FUNCTION_BLOCK T_SubModuleCollection EXTENDS T_CollectionBase

METHOD PUBLIC AddModule : BOOL
VAR_INPUT
  newModule : I_PackML_BaseModule;
END_VAR
VAR
	item : I_InterfaceBase;
END_VAR
IF newModule = 0 THEN
	LogError( 'Cannot AddModule invalid ref' );
	RETURN;
END_IF

IF NOT __QUERYINTERFACE(newModule, item) THEN
	LogError( 'Cannot AddModule  NOT __QUERYINTERFACE(newComponent, item)' );
	RETURN;
END_IF

IF HasItem( item := item ) THEN
	LogWarning( 'Module already in collection.' );
	RETURN;
END_IF

AddModule := addInSpareSlot( item := item );
END_METHOD

METHOD PUBLIC AllInAskedState : BOOL
VAR_INPUT
	State : Tc3_PackML_V2.E_PMLState;
END_VAR
VAR
	i : UDINT;
	Module : I_PackML_BaseModule;
	item : I_InterfaceBase;
END_VAR
IF Count = 0 THEN
	AllInAskedState := TRUE;
	RETURN;
END_IF

FOR i := 0 TO Count -1 DO

	IF NOT 	TryGetItem(i, item => item) THEN
		RETURN;
	END_IF
	
	IF NOT __QUERYINTERFACE(item, Module) THEN
		RETURN;
	END_IF
		
	IF Module.CurrentState <> State THEN
		RETURN;
	END_IF
		
END_FOR

AllInAskedState := TRUE;
END_METHOD

PROPERTY AnyError : BOOL
GET
VAR
  i : UDINT;
  Module : I_PackML_BaseModule;
  item : I_InterfaceBase;
 END_VAR
IF Count = 0 THEN
  RETURN;
END_IF

FOR i := 0 TO Count -1 DO

	IF NOT 	TryGetItem(i, item => item) THEN
		RETURN;
	END_IF
	
	IF NOT __QUERYINTERFACE(item, Module) THEN
		RETURN;
	END_IF
		
	IF Module.Error THEN
		AnyError := TRUE;
		RETURN;
	END_IF

END_FOR
END_GET
END_PROPERTY

METHOD PUBLIC AnyInAskedState : BOOL
VAR_INPUT
	State : Tc3_PackML_V2.E_PMLState;
END_VAR
VAR_OUTPUT
	Module : I_PackML_BaseModule;	
END_VAR
VAR
	i : UDINT;

	item : I_InterfaceBase;
END_VAR
IF Count = 0 THEN
	RETURN;
END_IF

FOR i := 0 TO Count -1 DO

	IF NOT 	TryGetItem(i, item => item) THEN
		RETURN;
	END_IF
	
	IF NOT __QUERYINTERFACE(item, Module) THEN
		RETURN;
	END_IF
		
	IF Module.CurrentState = State THEN
		AnyInAskedState := TRUE;
		RETURN;
	END_IF
		
END_FOR
END_METHOD

METHOD CyclicLogic
VAR
  i : UDINT;
  Module : I_PackML_BaseModule;
  item : I_InterfaceBase;
END_VAR
IF Count = 0 THEN
  RETURN;
END_IF

FOR i := 0 TO Count -1 DO
	TryGetItem(i, item => item);
	__QUERYINTERFACE(item, Module);
	IF Module <> 0 THEN
  		Module.CyclicLogic();
	END_IF	
END_FOR
END_METHOD

PROPERTY PUBLIC InitialisedAll : BOOL
GET
VAR
  i : UDINT;
  Module : I_PackML_BaseModule;
  item : I_InterfaceBase;
 END_VAR
IF Count = 0 THEN
	InitialisedAll := TRUE;
  RETURN;
END_IF

FOR i := 0 TO Count -1 DO

	IF NOT 	TryGetItem(i, item => item) THEN
		RETURN;
	END_IF
	
	IF NOT __QUERYINTERFACE(item, Module) THEN
		RETURN;
	END_IF
		
	IF NOT Module.InitComplete THEN
		RETURN;
	END_IF
		

END_FOR

InitialisedAll := TRUE;
END_GET
END_PROPERTY

METHOD PUBLIC NotifyModeChanged
VAR_INPUT
    Mode : E_PMLUnitMode;
END_VAR
VAR
	i : UDINT;
	Module : I_PackML_BaseModule;
	item : I_InterfaceBase;
END_VAR
IF Count = 0 THEN
  RETURN;
END_IF

FOR i := 0 TO Count -1 DO

	IF NOT 	TryGetItem(i, item => item) THEN
		RETURN;
	END_IF
	
	IF NOT __QUERYINTERFACE(item, Module) THEN
		RETURN;
	END_IF
		
	Module.ChangeMode(Mode);
		
END_FOR
END_METHOD

METHOD PUBLIC NotifyStateChanged
VAR_INPUT
	CommandedState : Tc3_PackML_V2.E_PMLCommand;
END_VAR
VAR
	i : UDINT;
	Module : I_PackML_BaseModule;
	item : I_InterfaceBase;
END_VAR
IF Count = 0 THEN
  RETURN;
END_IF

FOR i := 0 TO Count -1 DO

	IF NOT 	TryGetItem(i, item => item) THEN
		RETURN;
	END_IF
	
	IF NOT __QUERYINTERFACE(item, Module) THEN
		RETURN;
	END_IF
		
	Module.ChangeState(CommandedState);
		
END_FOR
END_METHOD

METHOD PUBLIC SetPMLSubModuleInfoActive : BOOL
VAR_IN_OUT
	SubModuleInfoArray : ARRAY[*] OF ST_PMLSubUnitInfo;
END_VAR
VAR
	i : DINT;
	lowerBound, upperBound : DINT;
END_VAR
lowerBound := LOWER_BOUND(SubModuleInfoArray,1);
upperBound := UPPER_BOUND(SubModuleInfoArray,1);

IF Count > upperBound THEN
	LogError('Can not SetPMLSubModuleInfoActive as  Count > upperBound');
	RETURN;
END_IF 

FOR i := lowerBound TO Count DO
    SubModuleInfoArray[i].Active := TRUE;
END_FOR;

SetPMLSubModuleInfoActive := TRUE;
END_METHOD

METHOD PUBLIC SetSubModuleInfoState
VAR_IN_OUT
	SubModuleInfoArray : ARRAY[*] OF ST_PMLSubUnitInfo;
END_VAR
VAR
	i : DINT;
	lowerBound, upperBound : DINT;
	Module : I_PackML_BaseModule;
	item : I_InterfaceBase;
END_VAR
lowerBound := LOWER_BOUND(SubModuleInfoArray,1);
upperBound := UPPER_BOUND(SubModuleInfoArray,1);

IF lowerBound <> 1 THEN
	RETURN;
END_IF

IF Count > upperBound THEN
	LogError('Can not SetPMLSubModuleInfoActive as  Count > upperBound');
	RETURN;
END_IF 



FOR i := 0 TO Count -1 DO

	IF NOT 	TryGetItem(i, item => item) THEN
		RETURN;
	END_IF
	
	IF NOT __QUERYINTERFACE(item, Module) THEN
		RETURN;
	END_IF
		
	 SubModuleInfoArray[i+1].eState :=  Module.CurrentState;
		
END_FOR
END_METHOD

METHOD PUBLIC StateReset
VAR
	i : UDINT;
	Module : I_PackML_BaseModule;
	item : I_InterfaceBase;
END_VAR
IF Count = 0 THEN
  RETURN;
END_IF

FOR i := 0 TO Count -1 DO

	IF NOT 	TryGetItem(i, item => item) THEN
		RETURN;
	END_IF
	
	IF NOT __QUERYINTERFACE(item, Module) THEN
		RETURN;
	END_IF
		
	IF Module.CurrentState = ePMLState_Stopped OR Module.CurrentState = ePMLState_Complete THEN
		Module.ChangeState (ePMLCommand_Reset);
	ELSIF Module.CurrentState = ePMLState_Aborted THEN
		Module.ChangeState (ePMLCommand_Clear);
	ELSIF Module.CurrentState = ePMLState_Clearing OR Module.CurrentState = ePMLState_Stopping OR Module.CurrentState = ePMLState_Resetting OR
		 Module.CurrentState = ePMLState_Idle THEN
		;
	ELSE
		Module.ChangeState(ePMLCommand_Abort);
	END_IF
		
END_FOR
END_METHOD

METHOD TryGetModule: BOOL
VAR_INPUT
	index : UDINT;
END_VAR
VAR_OUTPUT
	Module : I_PackML_BaseModule;
END_VAR
VAR
	item : I_InterfaceBase;
END_VAR
IF NOT SUPER^.TryGetItem(index := index, item => item) THEN
	LogError( 'Cannot TryGetComponent NOT SUPER^.TryGetItem(index := index, item => item) ' );
	RETURN;
END_IF

IF NOT __QUERYINTERFACE(item, Module) THEN
	LogError( 'Cannot TryGetComponent   NOT __QUERYINTERFACE(item, Module) ' );
	RETURN;
END_IF

TryGetModule := Module <> 0;
END_METHOD

END_FUNCTION_BLOCK

(* stored: Version 1.1.0.1, ProductVersion 3.1.4024.12
   POU T_SubModuleCollection: Id {e452d146-811c-4c16-9bd5-d9b031d0f126}, SpecialFunc None
   Method AddModule: Id {53fec14b-7f0d-4c8d-b489-4f8a2e7a91db}
   Method AllInAskedState: Id {c5525ce9-7897-4cf9-8030-5bde5f91a91f}
   Property AnyError: Id {eb31021d-4235-42c3-9509-05306c59aad0}
   Get Get: Id {5c9aadd3-4bed-46fd-99cb-3ec8209718e2}
   Method AnyInAskedState: Id {fd7aede1-97d0-4952-ae9a-bdb82589f7f4}
   Method CyclicLogic: Id {14da67f3-5fa4-4574-9988-115d51302eb8}
   Property InitialisedAll: Id {cb8be73b-6402-458a-bffd-aa60da85ce4b}
   Get Get: Id {5fb1c1d1-cf1d-4536-8532-22fb2763eeb1}
   Method NotifyModeChanged: Id {4b757abb-b5fa-4f69-8c19-ba1cf5b656bd}
   Method NotifyStateChanged: Id {4a22e1ac-0e21-4315-95e2-0fceb8c44e5e}
   Method SetPMLSubModuleInfoActive: Id {d86cc83d-fd36-40fc-bc91-98090402b698}
   Method SetSubModuleInfoState: Id {b0c8fd84-e58b-4bb0-93a5-199ec32b4722}
   Method StateReset: Id {f3e56b8e-4e67-469f-b002-8fff282ece26}
   Method TryGetModule: Id {6a10edd7-8fc0-4b22-9321-1adf10171732} *)
